FUNCTION_BLOCK ScriblyActuatorPen EXTENDS ZEquipment.ActuatorDigitalBiLsPlusMinus

METHOD PUBLIC DownAsync
VAR_INPUT
  startToken : ZCore.IStartToken;
END_VAR
MoveMinusAsync(startToken:=startToken);
END_METHOD

METHOD PUBLIC IsDown : BOOL
VAR_INPUT
END_VAR
IsDown := IsAtMinus();
END_METHOD

METHOD PUBLIC IsUp : BOOL
VAR_INPUT
END_VAR
IsUp := IsAtPlus();
END_METHOD

METHOD PUBLIC UpAsync
VAR_INPUT
  startToken : ZCore.IStartToken;
END_VAR
MovePlusAsync(startToken:=startToken);
END_METHOD

END_FUNCTION_BLOCK

(* stored: Version 1.1.0.1
   POU ScriblyActuatorPen: Id {4a720069-9d52-49a9-907c-8381652b91b3}, SpecialFunc None
   Method DownAsync: Id {16b7ebe7-9f3a-40ad-938b-b4397bebbd46}
   Method IsDown: Id {a17f2c38-789b-4ad9-a297-e5f1356dcdfc}
   Method IsUp: Id {ed5dba49-d072-4023-9805-135bf0833128}
   Method UpAsync: Id {4d589e7b-ce12-4a90-8abe-1fcba0cf22f7} *)
